// TIA Portal V20 export
TYPE "typePacOutputData"
// stored: Access Published
   STRUCT
      resetMax : Bool;   // Reset the maximum values
      resetMin : Bool;   // Reset the minimum values
      resetCounter : Bool;   // Reset the energy counters
      ackDiag : Bool;   // Acknowledge device diagnostics
      syncDemandPeriod : Bool;   // Synchronization of the demand period
      startStopProcessCounter : Bool;   // Process counter start/stop
      copyResetProcessCounter : Bool;   // Copy and reset process counter
      resetProcessCounter : Bool;   // Reset process counter
      switchHighTarif : Bool;   // Switch to high tarif (HT)
      switchLowTarif : Bool;   // Switch to low tarif (LT)
      switchOut_0 : Bool;   // Switch output 0.0: ON=1, OFF=0
      switchOut_1 : Bool;   // Switch output 0.1: ON=1, OFF=0
   END_STRUCT;
END_TYPE
